// TIA Portal V19 export
DATA_BLOCK "InputsToScada"   // DB16
{ S7_Optimized_Access := 'TRUE' }
AUTHOR : FLA
FAMILY : UHT
VERSION : 1.0
// stored: AutoNumber false, MemoryReserve 0
   VAR RETAIN
      dw0 : Int;   // Used by intouch for direct input I12.0 - I13.7
      dw2 : Int;   // Used by intouch for direct input I16.0 - I17.7
      dw4 : Int;   // Used by intouch for direct input I24.0 - I25.7
      dw6 : Int;   // Used by intouch for direct input I32.0 - I33.7
      dw8 : Int;   // Used by intouch for direct input I44.0 - I45.7
      dw10 : Int;   // Used by intouch for direct input I46.0 - I47.7
   END_VAR
BEGIN
END_DATA_BLOCK
